// TIA Portal V19 export
TYPE "LEXCHANGETRAY_typeHandlingXyzEm_toNgConveyorFeedback"
// stored: Access Published
   STRUCT
      transferEnable : Bool;   // 请求转移
      running : Bool;   // 放料中
   END_STRUCT;
END_TYPE
